INTERFACE I_1s_UPS

METHOD AcknowledgePowerFailDetect
VAR_INPUT
END_VAR
END_METHOD

PROPERTY bPowerFailDetect : BOOL
GET
END_GET
END_PROPERTY

PROPERTY bReady : BOOL
GET
END_GET
END_PROPERTY

PROPERTY e1sUpsState : E_S_UPS_State
GET
END_GET
END_PROPERTY

METHOD Execute
VAR_INPUT
END_VAR
END_METHOD

//FB_Init は常に暗黙的に使用可能で、主に初期化に使用されます。
//戻り値は評価されません。特定の結果を得るために、メソッドを明示的に宣言し、
//そのメソッドに標準の初期化コードをもったコードを追加することができます。戻り値を評価できます。
METHOD FB_Init: BOOL
VAR_INPUT
    bInitRetains: BOOL; // TRUE: 保持変数は初期化されます (ウォーム リセット、あるいはコールド リセット)
    bInCopyCode: BOOL;  // TRUE: 後でコードをコピーする (オンライン変更) ために、インスタンスをコピーします。

	PcAmsNetId					:AMSNETID;		//PC AMS Net ID
END_VAR
END_METHOD

END_INTERFACE

(* stored: Version 1.1.0.1
   Itf I_1s_UPS: Id {b4b1b3e2-fd93-4da2-92d1-453053502d99}
   Method AcknowledgePowerFailDetect: Id {81ddd59c-e5f7-453b-8714-ef4093d04315}
   Property bPowerFailDetect: Id {f8195a76-69b2-4f5a-93ed-cdcdf49a6394}
   Get Get: Id {92afdf7f-c298-4063-8ff0-c74db2a46fee}
   Property bReady: Id {292eb10e-6971-487f-b74b-4f1aecf9e276}
   Get Get: Id {262507eb-21c3-483f-bf8c-4fcfa1cb1278}
   Property e1sUpsState: Id {a73a48bb-8a97-4702-94a0-6f8e82e8979f}
   Get Get: Id {bdd0a802-9e7f-4583-9abb-873005299db7}
   Method Execute: Id {37908e70-6383-4f51-be8a-bdb845ca805c}
   Method FB_Init: Id {f38676ad-7c84-4fd7-bae1-539d65824671} *)
